FUNCTION_BLOCK FB_DifferentCVCamera EXTENDS FB_ActionBasic
VAR_INPUT
    xExecute    : BOOL;
    xAbort      : BOOL;
	xReset		: BOOL;
    Cylinder 	: REFERENCE TO UNI_CylinderList;
    TimeOut  	: LREAL := 600; // Unit : s
	Input		: ST_InputTable;
	OutPut		: ST_OutputTable;
	Motor		: REFERENCE TO UNI_MotorList;
	BoxCameraDone :BOOL;
END_VAR	
VAR_OUTPUT
    xAborted : BOOL;
    iErrorID : INT;
    ErrorMsg : STRING;
	UseBoxCamera	:BOOL;
END_VAR
VAR
    StateBehaviour   : CBML.ETrigATo;
    CurrentPosition : ST_PositionTable;
	uiCyclicStep    : UINT := 0;
	TON_DelaySensor	:TON;
	TON_TimeOut		:TON;
	TON_ArriviedTimeOut :TON ;
	TON_CameraTimeOut	:TON;
	TON_ConveyorTimeOut	:TON;
	Reset_Rtrig 	:R_TRIG;
	fbExecuteEdgeDetect :FB_EdgeDetect;
END_VAR

THIS^.IBehaviourModel := StateBehaviour;
StateBehaviour(xExecute := xExecute,
              xAbort := xAbort OR fbExecuteEdgeDetect.xFallingEdge,
              udiTimeOut := LREAL_TO_UDINT( TimeOut*1000000),
              xDone => xDone,
              xBusy => xBusy,
              xError => xError,
              xAborted => xAborted);
//Error Mes
iErrorID := StateBehaviour._model.iErrorID;
ErrorMsg := M_GetErrorMsg(xErrorID := iErrorID);  

//Make sure that C# turns off execute to shut down the service
fbExecuteEdgeDetect(xInput :=xExecute);

//Reset 
Reset_Rtrig(CLK:= xReset);
IF Reset_Rtrig.Q THEN
	StateBehaviour.ResetModel(xCommit:=xReset);
END_IF

//Action
A00_BaseUnits();

ACTION A00_BaseUnits:
TON_DelaySensor(PT:= T#1S);
TON_TimeOut(PT := T#20S);
TON_ArriviedTimeOut(PT:= T#60S);
TON_CameraTimeOut(PT :=T#250S);
TON_ConveyorTimeOut(PT :=T#60S);
END_ACTION

METHOD CleanupAction
VAR_INPUT
    xAbortProposed : BOOL;
    iErrorIDProposed: INT;
END_VAR
VAR_OUTPUT
    xComplete : BOOL := TRUE;
    xAbort: BOOL := xAbortProposed;
 	iErrorID : INT := iErrorIDProposed;
END_VAR
xComplete :=FALSE;
TON_DelaySensor.IN :=FALSE;
TON_TimeOut.IN := FALSE;
TON_ArriviedTimeOut.IN :=FALSE;
TON_CameraTimeOut.IN :=FALSE;
TON_ConveyorTimeOut.IN :=FALSE;

UseBoxCamera	:= FALSE;
BoxCameraDone	:= FALSE;

Cylinder.List.fbDifferentSizeCV_Block1.M_Retract();
Motor.List.TransmitDifferentSideCV.M_MotorStop();

IF Cylinder.List.fbDifferentSizeCV_Block1.InRearPosition AND 
	Motor.List.TransmitDifferentSideCV.InStopped THEN
	    xComplete := TRUE;
END_IF
END_METHOD

METHOD CyclicAction
VAR_INPUT
    itfTimingController : CBML.ITimingController;
END_VAR
VAR_OUTPUT
    xComplete : BOOL := TRUE;
    iErrorID : INT := 0;
END_VAR
VAR_INST
	bMoveConveyorForward	 : BOOL;
END_VAR
xComplete := FALSE;
IF bMoveConveyorForward THEN
	IF NOT Motor.List.TransmitDifferentSideCV.InBackWard THEN
		Motor.List.TransmitDifferentSideCV.M_MoveForward();
	END_IF
END_IF
CASE uiCyclicStep OF
    0:	//keep for use
	bMoveConveyorForward:=FALSE;
		uiCyclicStep :=1000;
		
	1000:	// block first box 
		TON_TimeOut.IN:=TRUE;
		//Cylinder.List.fbDifferentSizeCV_Press1.M_Retract();
		Cylinder.List.fbDifferentSizeCV_Block1.M_Extend();
		Cylinder.List.fbTransmitCV_CamaraHoriz.M_Extend();
		IF Cylinder.List.fbDifferentSizeCV_Block1.InFrontPosition AND 
			Cylinder.List.fbTransmitCV_CamaraHoriz.InFrontPosition (*AND
			Cylinder.List.fbDifferentSizeCV_Press1.InRearPosition*)  THEN
			TON_TimeOut.IN:=FALSE;
			uiCyclicStep :=1050;
		END_IF
		IF TON_TimeOut.Q THEN
			iErrorID := 7;
		END_IF
//	1025:	//check box on sensor
//		IF Input.bDifferentSizeCV_BoxDetect2_Sensor THEN
//			Motor.List.TransmitDifferentSideCV.M_MoveBackward();
//			uiCyclicStep :=1030;
//		ELSE
//			uiCyclicStep :=1050;
//		END_IF
//	1030:		//check box leave sensor
//		IF NOT Input.bDifferentSizeCV_BoxDetect2_Sensor	THEN
//			bMoveConveyorForward:=FALSE;
//			Motor.List.TransmitDifferentSideCV.M_MotorStop();
//			uiCyclicStep :=1040;
//		END_IF
//	1040:		//Check motor stop
//		IF Motor.List.TransmitDifferentSideCV.InStopped THEN
//			uiCyclicStep := 1050;
//		END_IF
		
	1050:	//motor moveforward
		TON_ConveyorTimeOut.IN:=TRUE;
		bMoveConveyorForward:=TRUE;
		Cylinder.List.fbDifferentSizeCV_Press1.M_Retract();
		//Motor.List.TransmitDifferentSideCV.M_MoveForward();
		IF 	Motor.List.TransmitDifferentSideCV.InForWard AND 
			Cylinder.List.fbDifferentSizeCV_Press1.InRearPosition	THEN
			TON_ConveyorTimeOut.IN:= FALSE;
			uiCyclicStep :=1100;
		END_IF
		IF TON_ConveyorTimeOut.Q THEN
			iErrorID := 7;
		END_IF
	1100:	//check first box arrive block
		TON_ArriviedTimeOut.IN:=TRUE;
		TON_DelaySensor.IN:=Input.bDifferentSizeCV_BoxDetect2_Sensor;
		IF TON_DelaySensor.Q THEN
			TON_DelaySensor.IN :=FALSE;
			TON_ArriviedTimeOut.IN :=FALSE;
			Cylinder.List.fbDifferentSizeCV_Press1.M_Extend();
			bMoveConveyorForward:=FALSE	;
			Motor.List.TransmitDifferentSideCV.M_MotorStop();
			uiCyclicStep :=1200;
		END_IF
		IF TON_ArriviedTimeOut.Q THEN
			iErrorID := 8;
		END_IF
		
	1200:	//send use camera & hold sencond box
		TON_ConveyorTimeOut.IN:=TRUE;	
		IF Cylinder.List.fbDifferentSizeCV_Press1.InFrontPosition AND
			Motor.List.TransmitDifferentSideCV.InStopped THEN
			TON_ConveyorTimeOut.IN:= FALSE;
			UseBoxCamera :=TRUE;			//send request
			uiCyclicStep :=1300;
		END_IF
		IF TON_ConveyorTimeOut.Q THEN
			iErrorID := 9 ;
		END_IF
		
	1300:	//Check C# send camera done
		TON_CameraTimeOut.IN:=TRUE;
		IF BoxCameraDone THEN
			TON_CameraTimeOut.IN :=FALSE;
			Cylinder.List.fbDifferentSizeCV_Block1.M_Retract();
			bMoveConveyorForward:=TRUE;
			//Motor.List.TransmitDifferentSideCV.M_MoveForward();
			uiCyclicStep :=1400;
		END_IF
		IF TON_CameraTimeOut.Q THEN 
			iErrorID :=10;
			//xAbort:=TRUE;				//abort resume C# checkBoxCameraDone FeedBack
		END_IF
		
	1400:	//First Box cross detect1 sensor
		TON_TimeOut.IN :=TRUE;
		IF Input.bDifferentSizeCV_BoxDetect1_Sensor THEN
			TON_TimeOut.IN :=FALSE;
			uiCyclicStep :=1500;
		END_IF
		IF TON_TimeOut.Q THEN
			iErrorID :=11;
		END_IF
		
	1500:	//cross sensor stop motor
		TON_DelaySensor.IN:=TRUE;
		IF NOT Input.bDifferentSizeCV_BoxDetect1_Sensor THEN
			TON_DelaySensor.IN:=FALSE;
			bMoveConveyorForward:=FALSE;
			Motor.List.TransmitDifferentSideCV.M_MotorStop();
			uiCyclicStep :=1600;
		END_IF
		IF TON_DelaySensor.Q THEN
			TON_DelaySensor.IN:=FALSE;
			bMoveConveyorForward:=FALSE;
			Motor.List.TransmitDifferentSideCV.M_MotorStop();
			uiCyclicStep :=1600;
		END_IF
	
	1600:	// wait motor stop 
		IF Motor.List.TransmitDifferentSideCV.InStopped THEN
			//Cylinder.List.fbDifferentSizeCV_Press1.M_Retract();
//			uiCyclicStep:=1700;
				xComplete :=TRUE;
		END_IF
	1700:	//make sure sencond box still 
//		IF Cylinder.List.fbDifferentSizeCV_Press1.InRearPosition THEN
//			xComplete :=TRUE;
//		END_IF
			
END_CASE
END_METHOD

METHOD ExitAction
VAR_INPUT
    xAfterCleanup : BOOL;
    xInCopyCode : BOOL;
END_VAR
END_METHOD

METHOD M_GetErrorMsg : T_MaxString
VAR_INPUT
	xErrorID: INT;
END_VAR

VAR
	
END_VAR
CASE xErrorID OF
	0:
		M_GetErrorMsg := 'No Error';
	1:
		M_GetErrorMsg := 'Action time out';
	2:
		M_GetErrorMsg := 'Position Data invalid';
///
	3:
		M_GetErrorMsg := 'Block1 cylinder not ready';
	4:
		M_GetErrorMsg := 'Press1 cylinder not ready';
	5:
		M_GetErrorMsg := 'CamaraHoriz cylinder not ready';
	6:
		M_GetErrorMsg := 'DifferentCV not ready ';
	7:	
		M_GetErrorMsg :=' Cylinder timeout';
	8:
		M_GetErrorMsg :='photo area have not box timeout';
	9:
		M_GetErrorMsg :='motor & cylinder timeout';
	10:
		M_GetErrorMsg :='C# BoxCameraDone timeout';
	11:
		M_GetErrorMsg :='Box cross sensor not detact timeout';
		
	20:
		M_GetErrorMsg :='Differnet conveyor full box infront';
END_CASE
END_METHOD

METHOD ResetAction
VAR_OUTPUT
    xComplete : BOOL := TRUE;
END_VAR
//IF xAbort THEN 
//	CASE uiCyclicStep OF 
//		1400:
//			uiCyclicStep :=1400;	
	
//	END_CASE
//END_IF
xComplete:= FALSE;
TON_DelaySensor.IN :=FALSE;
TON_TimeOut.IN := FALSE;
TON_ArriviedTimeOut.IN :=FALSE;
TON_CameraTimeOut.IN :=FALSE;
TON_ConveyorTimeOut.IN :=FALSE;
xComplete := TRUE;
END_METHOD

METHOD StartAction
VAR_OUTPUT
    xComplete : BOOL := TRUE;
	iErrorID : INT := 0;
END_VAR
xComplete :=FALSE;
TON_DelaySensor.IN :=FALSE;
TON_TimeOut.IN := FALSE;
TON_ArriviedTimeOut.IN :=FALSE;
TON_CameraTimeOut.IN :=FALSE;
TON_ConveyorTimeOut.IN :=FALSE;
uiCyclicStep :=0;
UseBoxCamera	:= FALSE;
BoxCameraDone	:= FALSE;

IF Input.bDifferentSizeCV_BoxDetect1_Sensor THEN
	iErrorID :=20;
END_IF

IF Cylinder.List.fbDifferentSizeCV_Block1.InRearPosition AND 
//	Cylinder.List.fbDifferentSizeCV_Press1.InRearPosition AND 		//Holding press make sure box cross behind
	//Cylinder.List.fbTransmitCV_CamaraHoriz.InRearPosition AND 
	Motor.List.TransmitDifferentSideCV.InStopped THEN
	    xComplete := TRUE;
END_IF


IF  Cylinder.List.fbDifferentSizeCV_Block1.xError  THEN
	iErrorID := 3; // Cylinder not ready
END_IF
IF  Cylinder.List.fbDifferentSizeCV_Press1.xError THEN
	iErrorID := 4; // Cylinder not ready
END_IF
IF  Cylinder.List.fbTransmitCV_CamaraHoriz.xError THEN
	iErrorID := 5;	//Cylinder not ready
END_IF
IF  Motor.List.TransmitDifferentSideCV.xError THEN
	iErrorID := 6;	//Conveyor not ready
END_IF
END_METHOD

END_FUNCTION_BLOCK

(* stored: Version 1.1.0.1, ProductVersion 3.1.4024.13
   POU FB_DifferentCVCamera: Id {f4ab733a-15a9-490a-bf47-b810290f7ccc}, SpecialFunc None
   Folder Action: Id {50b7549f-3c45-4ccf-a4a7-1cdf3c96151f}
   Action A00_BaseUnits: Id {ecb63a04-5545-4c1d-8290-f4ae59068027}
   Method CleanupAction: Id {84d205e3-84a9-4e6e-91e2-34f7af845f9a}
   Method CyclicAction: Id {dd093b31-2fe3-4187-9bd9-74b44ab660f6}
   Method ExitAction: Id {249c6dab-8479-4fb7-ad51-11e60e594e10}
   Method M_GetErrorMsg: Id {07171412-48bc-4271-a493-d60c93b6db04}
   Method ResetAction: Id {bbc4d767-cb94-4960-954c-a81bc8ad836f}
   Method StartAction: Id {d5f673ab-d024-4521-94fc-f22c207174d7} *)
